// TIA Portal V18 export
// export: Created 2026-06-12T02:00:00Z, ExportSetting WithDefaults
VAR_GLOBAL   // PLC tag table "PLC_Tags_B3to7"
   Timer_Sim_Pulse_Output AT %M1210.0 : Bool;   // Xung 50ms cho simulation
   Sim_Dir AT %M1210.1 : Bool;   // Hướng đếm: 0=Tăng, 1=Giảm
   Sim_Counter AT %MD1200 : Real;   // Bộ đếm 0-100 cho simulation
   Sim_Val_Norm AT %MD1204 : Real;   // Giá trị chuẩn hóa 0.0-1.0
   AI_B3_Sequence_Count AT %MD0 : Real;   // 0-100
   AI_B3_Flow_CIP_Center AT %MD4 : Real;   // 100-200 L/h
   AI_B3_Temp_CIP_Upper AT %MD8 : Real;   // 50-80 °C
   AI_B3_Pressure_CIP_1 AT %MD12 : Real;   // 7.0-8.0 bar
   AI_B3_Temp_Chaff_1 AT %MD16 : Real;   // 50-80 °C
   AI_B3_Flow_CIP_Feed AT %MD20 : Real;   // 100-200 L/h
   AI_B3_Temp_Steam_1 AT %MD24 : Real;   // 50-80 °C
   AI_B3_Flow_UCWW_1 AT %MD28 : Real;   // 100-200 L/h
   AI_B3_RPM_Screw_Conv AT %MD32 : Real;   // 800-1200 RPM
   AI_B3_Temp_Condensate_1 AT %MD36 : Real;   // 50-80 °C
   AI_B3_Pressure_Screw_1 AT %MD40 : Real;   // 7.0-8.0 bar
   AI_B3_Flow_CWW_Out AT %MD44 : Real;   // 100-200 L/h
   AI_B3_Pressure_CWW_1 AT %MD48 : Real;   // 7.0-8.0 bar
   AI_B3_Temp_Decanter2 AT %MD52 : Real;   // 50-80 °C
   AI_B3_RPM_Rotary2 AT %MD56 : Real;   // 800-1200 RPM
   AI_B3_RPM_Rotary1 AT %MD60 : Real;   // 800-1200 RPM
   AI_B3_Temp_GroundSilo AT %MD64 : Real;   // 50-80 °C
   AI_B3_Flow_GroundSilo AT %MD68 : Real;   // 100-200 L/h
   AI_B3_Pressure_Mid_1 AT %MD72 : Real;   // 7.0-8.0 bar
   AI_B3_Flow_Condensate AT %MD76 : Real;   // 100-200 L/h
   AI_B3_Flow_Sump_Out AT %MD80 : Real;   // 100-200 L/h
   AI_B3_Level_Sump AT %MD84 : Real;   // 30-80 %
   AI_B3_Pressure_Decant1 AT %MD88 : Real;   // 7.0-8.0 bar
   AI_B3_Pressure_Decant2 AT %MD92 : Real;   // 7.0-8.0 bar
   AI_B3_Flow_Decant1 AT %MD96 : Real;   // 100-200 L/h
   AI_B3_Temp_Decant1 AT %MD100 : Real;   // 50-80 °C
   AI_B3_Temp_FBB_Boiler AT %MD104 : Real;   // 50-80 °C
   AI_B3_Temp_CWW_Out AT %MD108 : Real;   // 50-80 °C
   AI_B3_Pressure_SUMP AT %MD112 : Real;   // 7.0-8.0 bar
   AI_B3_Flow_SUMP AT %MD116 : Real;   // 100-200 L/h
   AI_B3_Level_CWW AT %MD120 : Real;   // 30-80 %
   AI_B3_Temp_FBB_Out AT %MD124 : Real;   // 50-80 °C
   AI_B3_Pressure_FBB_Out AT %MD128 : Real;   // 7.0-8.0 bar
   AI_B3_Flow_FBB_Out AT %MD132 : Real;   // 100-200 L/h
   AI_B4_Daq_C AT %MD200 : Real;   // 0-100
   AI_B4_TPH_Total AT %MD204 : Real;   // 100-200 T/h
   AI_B4_KG_CM_Main AT %MD208 : Real;   // 7.0-8.0 kg/cm2
   AI_B4_DRM_LVL1 AT %MD212 : Real;   // 30-80 %
   AI_B4_DRM_LVL2 AT %MD216 : Real;   // 30-80 %
   AI_B4_MW_Output AT %MD220 : Real;   // 0-50 MW
   AI_B4_KG_CM_2 AT %MD224 : Real;   // 7.0-8.0 kg/cm2
   AI_B4_Hc_Value AT %MD228 : Real;   // 0-100
   AI_B4_Temp_AirHeater_In1 AT %MD232 : Real;   // 50-80 °C
   AI_B4_Temp_AirHeater_In2 AT %MD236 : Real;   // 50-80 °C
   AI_B4_Temp_AirHeater_In3 AT %MD240 : Real;   // 50-80 °C
   AI_B4_Temp_AirHeater_Out1 AT %MD244 : Real;   // 50-80 °C
   AI_B4_Temp_AirHeater_Out2 AT %MD248 : Real;   // 50-80 °C
   AI_B4_Pres_AH_mmWC_1 AT %MD252 : Real;   // 7.0-8.0 mmWC
   AI_B4_Pres_AH_mmWC_2 AT %MD256 : Real;   // 7.0-8.0 mmWC
   AI_B4_Pres_AH_Pct_1 AT %MD260 : Real;   // 20-80 %
   AI_B4_Temp_AH_Out3 AT %MD264 : Real;   // 50-80 °C
   AI_B4_Pres_FDH_mmWC AT %MD268 : Real;   // 7.0-8.0 mmWC
   AI_B4_RPM_PAF1 AT %MD272 : Real;   // 800-1200 RPM
   AI_B4_Pct_RPC308_SP AT %MD276 : Real;   // 20-80 %
   AI_B4_Pct_RPC308_PV AT %MD280 : Real;   // 20-80 %
   AI_B4_Pres_PAF1_mmWC AT %MD284 : Real;   // 7.0-8.0 mmWC
   AI_B4_Pct_FDF1_SP AT %MD288 : Real;   // 20-80 %
   AI_B4_Pct_FDF1_PV AT %MD292 : Real;   // 20-80 %
   AI_B4_Pct_FDF1_OUT AT %MD296 : Real;   // 20-80 %
   AI_B4_RPM_FDF1 AT %MD300 : Real;   // 800-1200 RPM
   AI_B4_Pct_RPC301_SP AT %MD304 : Real;   // 20-80 %
   AI_B4_Pct_RPC301_PV AT %MD308 : Real;   // 20-80 %
   AI_B4_Pct_RPC301_OUT AT %MD312 : Real;   // 20-80 %
   AI_B4_mA_ESP1 AT %MD316 : Real;   // 50-200 mA
   AI_B4_mA_ESP2 AT %MD320 : Real;   // 50-200 mA
   AI_B4_mA_ESP3 AT %MD324 : Real;   // 50-200 mA
   AI_B4_mA_ESP4 AT %MD328 : Real;   // 50-200 mA
   AI_B4_V_ESP1 AT %MD332 : Real;   // 0-400 V
   AI_B4_V_ESP2 AT %MD336 : Real;   // 0-400 V
   AI_B4_V_ESP3 AT %MD340 : Real;   // 0-400 V
   AI_B4_V_ESP4 AT %MD344 : Real;   // 0-400 V
   AI_B4_Pct_RPC305_SP AT %MD348 : Real;   // 20-80 %
   AI_B4_Pct_RPC305_PV AT %MD352 : Real;   // 20-80 %
   AI_B4_RPM_IDF1 AT %MD356 : Real;   // 800-1200 RPM
   AI_B4_Pct_RPC305_VFD AT %MD360 : Real;   // 20-80 %
   AI_B4_Pct_FDF2_SP AT %MD364 : Real;   // 20-80 %
   AI_B4_Pct_FDF2_PV AT %MD368 : Real;   // 20-80 %
   AI_B4_Pct_FDF2_OUT AT %MD372 : Real;   // 20-80 %
   AI_B4_RPM_FDF2 AT %MD376 : Real;   // 800-1200 RPM
   AI_B4_Pct_RPC306_SP AT %MD380 : Real;   // 20-80 %
   AI_B4_Pct_RPC306_PV AT %MD384 : Real;   // 20-80 %
   AI_B4_Pct_RPC306_OUT AT %MD388 : Real;   // 20-80 %
   AI_B4_RPM_IDF2 AT %MD392 : Real;   // 800-1200 RPM
   AI_B4_Pct_RPC306_VFD AT %MD396 : Real;   // 20-80 %
   AI_B4_Pres_FDF_mmWC AT %MD400 : Real;   // 7.0-8.0 mmWC
   AI_B4_TEST1_Value AT %MD404 : Real;   // 0-100
   AI_B4_Pct_PAF1_SP AT %MD408 : Real;   // 20-80 %
   AI_B4_Pct_PAF1_PV AT %MD412 : Real;   // 20-80 %
   AI_B4_Pres_PAF2_mmWC AT %MD416 : Real;   // 7.0-8.0 mmWC
   AI_B4_RPM_PAF2 AT %MD420 : Real;   // 800-1200 RPM
   AI_B4_Pct_RPC308b_SP AT %MD424 : Real;   // 20-80 %
   AI_B4_Pct_RPC308b_PV AT %MD428 : Real;   // 20-80 %
   AI_B4_Pct_DAM303B_SP AT %MD432 : Real;   // 20-80 %
   AI_B4_Pct_DAM304B_SP AT %MD436 : Real;   // 20-80 %
   AI_B5_CA_Fan_Motor_DE_Temp AT %MD500 : Real;   // 50-80 °C
   AI_B5_CA_Fan_Motor_NDE_Temp AT %MD504 : Real;   // 50-80 °C
   AI_B5_CA_Fan_DE_Temp AT %MD508 : Real;   // 50-80 °C
   AI_B5_CA_Fan_NDE_Temp AT %MD512 : Real;   // 50-80 °C
   AI_B5_CA_Fan_DE_Vib AT %MD516 : Real;   // 0-10 mm/s
   AI_B5_CA_Fan_NDE_Vib AT %MD520 : Real;   // 0-10 mm/s
   AI_B5_SP_700FN03 AT %MD524 : Real;   // 100-200 L/h
   AI_B5_SP_700HES01 AT %MD528 : Real;   // 100-200 L/h
   AI_B5_SP_700DA4 AT %MD532 : Real;   // 20-30 Hz
   AI_B5_SP_700DA6 AT %MD536 : Real;   // 20-30 Hz
   AI_B5_SP_700DA7 AT %MD540 : Real;   // 20-30 Hz
   AI_B5_SP_700FN2_DA1 AT %MD544 : Real;   // 20-30 Hz
   AI_B5_Sep_Motor_Top_Temp AT %MD548 : Real;   // 50-80 °C
   AI_B5_Sep_Bottom_Bear_Temp AT %MD552 : Real;   // 50-80 °C
   AI_B5_Trend_Val_1 AT %MD556 : Real;   // 0-100 %
   AI_B5_Trend_Val_2 AT %MD560 : Real;   // 0-100 %
   AI_B5_Trend_Val_3 AT %MD564 : Real;   // 0-100 %
   AI_B5_700FN03_RPM AT %MD568 : Real;   // 800-1200 RPM
   AI_B5_700HES01_Flow AT %MD572 : Real;   // 100-200 L/h
   AI_B5_700FN10_Speed AT %MD576 : Real;   // 20-30 Hz
   AI_B5_700CM01_Current AT %MD580 : Real;   // 50-200 A
   AI_B5_Lub_Stop_Time AT %MD584 : Real;   // 0-300 Sec
   AI_B5_Main_Drive_ReHealth AT %MD588 : Real;   // 0-300 Sec
   AI_B5_CM_LRS_IN AT %MD592 : Real;   // 50-80 °C
   AI_B5_CM_LRS_OUT AT %MD596 : Real;   // 50-80 °C
   AI_B5_CM_Mill_Oil_Temp AT %MD600 : Real;   // 50-80 °C
   AI_B5_CM_OilTrun_BER_Temp AT %MD604 : Real;   // 50-80 °C
   AI_B5_CM_OilTrun_BER2_Temp AT %MD608 : Real;   // 50-80 °C
   AI_B5_CM_OilPinion_BER_Temp AT %MD612 : Real;   // 50-80 °C
   AI_B5_CM_GB_IL_Shaft_BER AT %MD616 : Real;   // 50-80 °C
   AI_B5_CM_Running_Hours AT %MD620 : Real;   // 0-8760 Hr
   AI_B5_CM_PS1_1_KG AT %MD624 : Real;   // 7-8 bar
   AI_B5_CM_PS1_2_KG AT %MD628 : Real;   // 7-8 bar
   AI_B5_NIBS_Value AT %MD632 : Real;   // 50-200 A
   AI_B5_800DC1_Temp AT %MD636 : Real;   // 50-80 °C
   AI_B5_800DC2_Temp AT %MD640 : Real;   // 50-80 °C
   AI_B5_800FN1_Speed AT %MD644 : Real;   // 20-30 Hz
   AI_B5_800FN2_Speed AT %MD648 : Real;   // 20-30 Hz
   AI_B5_800YF1_Flow AT %MD652 : Real;   // 100-200 L/h
   AI_B5_800YF2_Flow AT %MD656 : Real;   // 100-200 L/h
   AI_B5_Silo1_Level_Bar1 AT %MD660 : Real;   // 0-100 %
   AI_B5_Silo1_Level_Bar2 AT %MD664 : Real;   // 0-100 %
   AI_B5_Silo2_Level_Bar1 AT %MD668 : Real;   // 0-100 %
   AI_B5_Silo2_Level_Bar2 AT %MD672 : Real;   // 0-100 %
   AI_B5_700FN01_Speed AT %MD676 : Real;   // 20-30 Hz
   AI_B5_700FN02_Speed AT %MD680 : Real;   // 20-30 Hz
   AI_B5_700AS07_Speed AT %MD684 : Real;   // 20-30 Hz
   AI_B5_700AS08_Flow AT %MD688 : Real;   // 100-200 L/h
   AI_B5_700FN09_Speed AT %MD692 : Real;   // 20-30 Hz
   AI_B5_700SFM01_Speed AT %MD696 : Real;   // 20-30 Hz
   AI_B5_700DA1_Flow AT %MD700 : Real;   // 100-200 L/h
   AI_B5_700DA4_Flow AT %MD704 : Real;   // 100-200 L/h
   AI_B5_700DA6_Temp AT %MD708 : Real;   // 50-80 °C
   AI_B5_700DA7_Temp AT %MD712 : Real;   // 50-80 °C
   AI_B5_700BL1_Load AT %MD716 : Real;   // 50-200 A
   AI_B5_700BL2_Load AT %MD720 : Real;   // 50-200 A
   AI_B5_700AS9_Flow AT %MD724 : Real;   // 100-200 L/h
   AI_B5_700FN13_Speed AT %MD728 : Real;   // 20-30 Hz
   AI_B6_TICR211_Temp AT %MD800 : Real;   // 50-80 °C
   AI_B6_TICR210_Temp AT %MD804 : Real;   // 50-80 °C
   AI_B6_TICR201_Tank_Temp AT %MD808 : Real;   // 50-80 °C
   AI_B6_PT201_Pressure AT %MD812 : Real;   // 7.0-8.0 bar
   AI_B6_Ph201_pH AT %MD816 : Real;   // 6.0-8.0 pH
   AI_B6_ORP201_ORP AT %MD820 : Real;   // 20-80 %
   AI_B6_DPL101_Level AT %MD824 : Real;   // 100-500 L
   AI_B6_TICR214_Temp AT %MD828 : Real;   // 50-80 °C
   AI_B6_TICR204_Temp AT %MD832 : Real;   // 50-80 °C
   AI_B6_TICR205_Temp AT %MD836 : Real;   // 50-80 °C
   AI_B6_TICR206_Temp AT %MD840 : Real;   // 50-80 °C
   AI_B6_FHC203_Flow AT %MD844 : Real;   // 100-200 L/h
   AI_B6_BPC201_Pressure AT %MD848 : Real;   // 7.0-8.0 bar
   AI_B7_K03_PT02_Pressure AT %MD900 : Real;   // 7-8 bar
   AI_B7_K03_TT04_Temp AT %MD904 : Real;   // 50-80 °C
   AI_B7_K03_TT05_Temp AT %MD908 : Real;   // 50-80 °C
   AI_B7_K03_TT06_Temp AT %MD912 : Real;   // 50-80 °C
   AI_B7_K03_TT07_Temp AT %MD916 : Real;   // 50-80 °C
   AI_B7_K03_PT07_Pressure AT %MD920 : Real;   // 7-8 bar
   AI_B7_K03_FT03_Flow AT %MD924 : Real;   // 100-200 L/h
   AI_B7_K03_Density_1 AT %MD928 : Real;   // 800-1000 kg/m3
   AI_B7_K03_LT01_Level AT %MD932 : Real;   // 20-80 cm
   AI_B7_K03_LT02_Level AT %MD936 : Real;   // 20-80 cm
   AI_B7_K03_TT01_Temp AT %MD940 : Real;   // 50-80 °C
   AI_B7_K03_TT02_Temp AT %MD944 : Real;   // 50-80 °C
   AI_B7_Reboiler_PV AT %MD948 : Real;   // 100-200 L/h
   AI_B7_Reboiler_SP AT %MD952 : Real;   // 100-200 L/h
   AI_B7_Reboiler_CV AT %MD956 : Real;   // 20-80 %
   AI_B7_HE03_Primary_Temp AT %MD960 : Real;   // 50-80 °C
   AI_B7_HE03_Secondary_Temp AT %MD964 : Real;   // 50-80 °C
   AI_B7_K03_L08_Level AT %MD968 : Real;   // 20-80 cm
   AI_B7_K03_L06_Level AT %MD972 : Real;   // 20-80 cm
   AI_B7_K03_L05_Level AT %MD976 : Real;   // 20-80 cm
   AI_B7_K03_L07_Level AT %MD980 : Real;   // 20-80 cm
   AI_B7_K03_L04_Level AT %MD984 : Real;   // 20-80 cm
   AI_B7_K03_L03_Level AT %MD988 : Real;   // 20-80 cm
   AI_B7_V03A_Density AT %MD992 : Real;   // 800-1000 kg/m3
   AI_B7_Kettle_Flow_SP AT %MD996 : Real;   // 100-200 kg/h
   AI_B7_Keboiler_Flow_SP AT %MD1000 : Real;   // 100-200 kg/h
   AI_B7_Reflux_Time_SP AT %MD1004 : Real;   // 0-60 Min
   AI_B7_Time_Remain AT %MD1008 : Real;   // 0-60 Min
   AI_B7_RD_Level_SP AT %MD1012 : Real;   // 20-80 cm
   AI_B7_Reflux_Flow_SP AT %MD1016 : Real;   // 100-200 L/h
   AI_B7_Collection_SP AT %MD1020 : Real;   // 100-200 L/h
   AI_B7_Total_Flowrate AT %MD1024 : Real;   // 100-200 L/h
   AI_B7_ML_Qty_SP AT %MD1028 : Real;   // 0-600 L
   AI_B7_ML_Qty_Total AT %MD1032 : Real;   // 0-600 L
   AI_B7_Material_Code AT %MD1036 : Real;   // 0-99
   AI_B7_Stage_Number AT %MD1040 : Real;   // 0-20
   AI_B7_Batch_Number AT %MD1044 : Real;   // 0-9999
   AI_B7_Current_User_ID AT %MD1048 : Real;   // 0-999
   AI_B7_K_05_L_704_HI AT %MD1052 : Real;   // 20-80 cm
   AI_B7_Density_SP AT %MD1056 : Real;   // 800-1000 kg/m3
   AI_B7_CTS_Flow_1 AT %MD1060 : Real;   // 100-200 kg/h
   AI_B7_CTS_Flow_2 AT %MD1064 : Real;   // 100-200 kg/h
   AI_B7_Steam_PT01_Temp AT %MD1068 : Real;   // 50-80 °C
   AI_B7_Steam_PT02_Temp AT %MD1072 : Real;   // 50-80 °C
   AI_B7_CWS_TT01_Temp AT %MD1076 : Real;   // 50-80 °C
   AI_B7_CWS_TT02_Temp AT %MD1080 : Real;   // 50-80 °C
   AI_B7_CWS_TT03_Temp AT %MD1084 : Real;   // 50-80 °C
   AI_B7_CWAR_TT01_Temp AT %MD1088 : Real;   // 50-80 °C
   AI_B7_CWAR_TT02_Temp AT %MD1092 : Real;   // 50-80 °C
   AI_B7_CWAR_TT03_Temp AT %MD1096 : Real;   // 50-80 °C
   AI_B7_CWAR_TT04_Temp AT %MD1100 : Real;   // 50-80 °C
   AI_B7_K03_CV01_PV AT %MD1104 : Real;   // 20-80 %
   AI_B7_K03_CV01_SP AT %MD1108 : Real;   // 20-80 %
   AI_B7_K03_CV01_CV AT %MD1112 : Real;   // 20-80 %
   AI_B7_Steam_CV01_PV AT %MD1116 : Real;   // 20-80 %
   AI_B7_Steam_CV01_SP AT %MD1120 : Real;   // 20-80 %
   AI_B7_Steam_CV01_CV AT %MD1124 : Real;   // 20-80 %
   AI_B7_K03_Jacket_PV AT %MD1128 : Real;   // 50-80 °C
   AI_B7_K03_Jacket_SP AT %MD1132 : Real;   // 50-80 °C
   AI_B7_K03_Jacket_CV AT %MD1136 : Real;   // 20-80 %
   AI_B7_CHWR_TT01_Temp AT %MD1140 : Real;   // 50-80 °C
   AI_B7_CHWR_TT02_Temp AT %MD1144 : Real;   // 50-80 °C
   AI_B7_CHWS_TT01_Temp AT %MD1148 : Real;   // 50-80 °C
   AI_B7_CHWS_TT02_Temp AT %MD1152 : Real;   // 50-80 °C
   AI_B7_K03_TT03_Temp AT %MD1156 : Real;   // 50-80 °C
END_VAR
